{attribute 'qualified_only'}
VAR_GLOBAL CONSTANT
    (* Some constants declared until dynamic arrays/vectors have been implemented *)
    MaxAmountOfTestSuites : UINT := 300;
    MaxAmountOfTestsForEachTestSuite : UINT := 100;
    MaxAmountOfAsserts : UINT := 300;
END_VAR

(* stored: Version 1.1.0.1, ProductVersion 3.1.4022.18
   GVL GVL_Constants_TcUnit: Id {798c1086-367a-4b55-afbc-d1cf17a88bb1} *)
